KUKA KRL program: ps_604res_c1_orig.src, ps_604res_c1_orig.dat

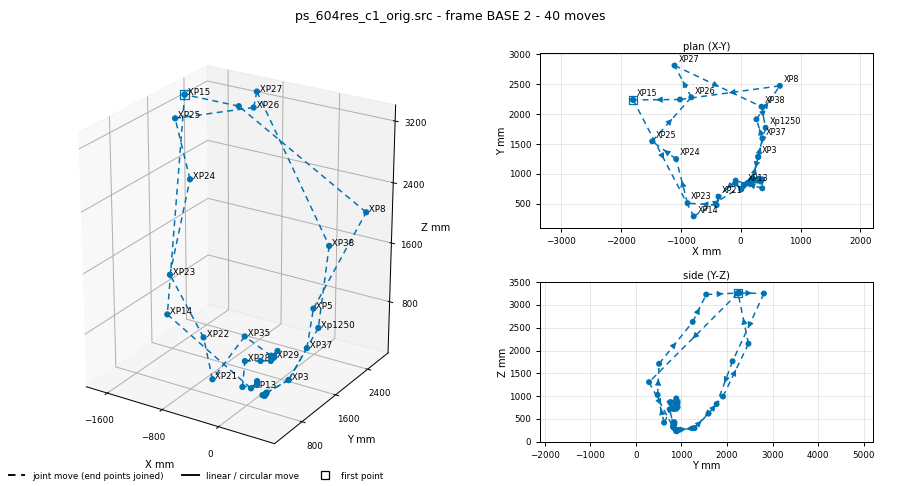
[picture p0: tool path of ps_604res_c1_orig.src in frame BASE 2, 40 of 40 moves have a stored position in this frame; points joined in program order, loops and branches not executed]
--- ps_604res_c1_orig.src ---
&ACCESS RVO
&COMMENT Solda Respot Accelo
DEF ps_604res_c1_orig( )
EXT e_Fraes1 ( )
EXT f_Fraes1 ( )
  ;FOLD INI;%{PE}%V2.2.2,%MKUKATPBASIS,%CINIT,%VCOMMON,%P
  ;FOLD BAS INI;%{PE}%V2.2.2,%MKUKATPBASIS,%CINIT,%VINIT,%P
  INTERRUPT DECL 3 WHEN $STOPMESS==TRUE DO IR_STOPM ( )
  INTERRUPT ON 3
  BAS (#INITMOV,0 )
  ;ENDFOLD
  ;FOLD A20 INI;%{E}%V2.2.2,%MKUKATPA20,%CINIT,%VINIT,%P
  IF ARC20==TRUE THEN
    A20 (ARC_INI)
    INTERRUPT DECL 6 WHEN $CYCFLAG[3]==FALSE DO A20(TECH_STOP2)
  ENDIF
  ;ENDFOLD
  ;FOLD A10 INI;%{E}%V2.2.2,%MKUKATPARC,%CINIT,%VINIT,%P
  IF A10_OPTION==#ACTIVE THEN
    INTERRUPT DECL 4 WHEN $CYCFLAG[2]==FALSE DO A10 (#APPL_ERROR)
    INTERRUPT DECL 7 WHEN A_ARC_SWI==#ACTIVE DO A10 (#ARC_SEAM)
    INTERRUPT DECL 5 WHEN A_FLY_ARC==TRUE DO A10 (#HPU_ARC)
    INTERRUPT  ON 5
    A10_INI ( )
  ENDIF
  ;ENDFOLD
  ;FOLD GRIPPER INI;%{E}%V2.2.2,%MKUKATPGRIPPER,%CINIT,%VINIT,%P
  USER_GRP(0,DUMMY,DUMMY,GDEFAULT)
  ;ENDFOLD
  ;FOLD SPOT INI;%{E}%V.2.2,%MKUKATPSPOT,%CINIT,%VINIT,%P
  USERSPOT(#INIT)
  ;ENDFOLD
  ;FOLD TOUCHSENSE INI;%{E}%V2.2.2,%MKUKATPTS,%CINIT,%VINIT,%P
  IF H70_OPTION THEN
    INTERRUPT DECL 15 WHEN $MEAS_PULSE[TOUCH_I[TOUCH_ACTIVE].IN_NR] DO H70 (6,CD0 )
    INTERRUPT DECL 16 WHEN $ZERO_MOVE DO H70 (7,CD0 )
    INTERRUPT DECL 17 WHEN $TECHPAR_C[FG_TOUCH,8]>0.5 DO H70 (8,CD0)
    H70 (1,CD0 )
  ENDIF
  ;ENDFOLD
  ;FOLD USER INI;%{P}%V2.2.2,%MKUKATPUSER,%CINIT,%VINIT,%P
  ;Make your modifications here
  ;ENDFOLD
  ;ENDFOLD

; Caracterização dos meios de produção: P13.060-R4
; Versão atual: 20/07/2013 12:00  Nome: Solda Respot Accelo
; Change: C1

chk_w1_wechs_ok ( )     ; VERIFICAÇÃO DE FERRAMENTA: C1

;FOLD Kollision.Ueberwachung_2_Ein ;%{PE}%MKUKATPUSER
COLLSTOP( 2, 1 ) ;INTERRUPTUEBERWACHT
;ENDFOLD

;FOLD PTP P15 CONT Vel= 80 % PDAT15 Tool[1]:GUN C1 Base[2]:Accelo;%{PE}%R 4.1.16,%MKUKATPBASIS,%CMOVE,%VPTP,%P 1:PTP, 2:P15, 3:C_PTP, 5:80, 7:PDAT15
$BWDSTART = FALSE
PDAT_ACT=PPDAT15
BAS(#PTP_DAT)
FDAT_ACT=FP15
BAS(#FRAMES)
BAS(#VEL_PTP,80)
PTP XP15 C_PTP
;ENDFOLD

;FOLD OUT 838 'Solic. Lib. Soldar Respot Geo1'  State= TRUE ;%{PE}%R 4.1.16,%MKUKATPBASIS,%COUT,%VOUTX,%P 2:838, 3:'Solic. Lib. Soldar Respot Geo1', 5:TRUE, 6:
$OUT[838]=TRUE
;ENDFOLD
;FOLD WAIT FOR IN 846 'R4 Aguarda Lib soldar RES geo 11'  State= TRUE ;%{PE}%R 4.1.16,%MKUKATPBASIS,%CWAIT_FOR,%VWAIT_FOR,%P 1:0, 2:846, 3:'R4 Aguarda Lib soldar RES geo 11', 5:TRUE, 6:
WAIT FOR $IN[846]==TRUE
;ENDFOLD
;FOLD OUT 838 'Solic. Lib. Soldar Respot Geo1'  State= FALSE ;%{PE}%R 4.1.16,%MKUKATPBASIS,%COUT,%VOUTX,%P 2:838, 3:'Solic. Lib. Soldar Respot Geo1', 5:FALSE, 6:
$OUT[838]=FALSE
;ENDFOLD


;FOLD OUT 851 'Libera AGV'  State= FALSE ;%{PE}%R 4.1.16,%MKUKATPBASIS,%COUT,%VOUTX,%P 2:851, 3:'Libera AGV', 5:FALSE, 6:
$OUT[851]=FALSE
;ENDFOLD


;FOLD PTP P14 CONT Vel= 80 % PDAT14 Tool[1]:GUN C1 Base[2]:Accelo;%{PE}%R 4.1.16,%MKUKATPBASIS,%CMOVE,%VPTP,%P 1:PTP, 2:P14, 3:C_PTP, 5:80, 7:PDAT14
$BWDSTART = FALSE
PDAT_ACT=PPDAT14
BAS(#PTP_DAT)
FDAT_ACT=FP14
BAS(#FRAMES)
BAS(#VEL_PTP,80)
PTP XP14 C_PTP
;ENDFOLD
;FOLD PTP P13 CONT Vel= 80 % PDAT13 Tool[1]:GUN C1 Base[2]:Accelo;%{PE}%R 4.1.16,%MKUKATPBASIS,%CMOVE,%VPTP,%P 1:PTP, 2:P13, 3:C_PTP, 5:80, 7:PDAT13
$BWDSTART = FALSE
PDAT_ACT=PPDAT13
BAS(#PTP_DAT)
FDAT_ACT=FP13
BAS(#FRAMES)
BAS(#VEL_PTP,80)
PTP XP13 C_PTP
;ENDFOLD
;FOLD PTP P17 CONT Vel= 80 % PDAT17 Tool[1]:GUN C1 Base[2]:Accelo;%{PE}%R 4.1.16,%MKUKATPBASIS,%CMOVE,%VPTP,%P 1:PTP, 2:P17, 3:C_PTP, 5:80, 7:PDAT17
$BWDSTART = FALSE
PDAT_ACT=PPDAT17
BAS(#PTP_DAT)
FDAT_ACT=FP17
BAS(#FRAMES)
BAS(#VEL_PTP,80)
PTP XP17 C_PTP
;ENDFOLD

;FOLD PTP SWP_62_0006 PDAT19 SPOT Gun= 1 RETR OPN PgNo1= 36 ACTIVE= 1 Tool[1]:GUN C1 Base[2]:Accelo;%{PE}%R 4.1.12,%MKUKATPSPOT,%CSPOT,%VPTP,%P 1:PTP, 2:SWP_62_0006, 3:, 5:80, 7:PDAT19, 10:1, 12:#FIRST, 14:#OPN, 16:36, 18:1, 20:0, 22:0, 24:1, 25:NORMAL
$BWDSTART = FALSE
PDAT_ACT=PPDAT19
BAS(#PTP_DAT)
FDAT_ACT=FSWP_62_0006
BAS(#FRAMES)
BAS(#VEL_PTP,PPDAT19.VEL)
S_ACT.GUN=1
S_ACT.PAIR=SDEFAULT.PAIR
S_ACT.RETR=#OPN
S_ACT.CLO_TM=1
S_ACT.PGNO1=36
S_ACT.PGNO2=SDEFAULT.PGNO2
S_ACT.PRESS1=SDEFAULT.PRESS1
S_ACT.PRESS2=SDEFAULT.PRESS2
S_READY=FALSE
PTP XSWP_62_0006
USERSPOT(#SPOT, S_ACT)
WAIT FOR S_READY
;ENDFOLD

;FOLD PTP P19 CONT Vel= 80 % PDAT20 Tool[1]:GUN C1 Base[2]:Accelo;%{PE}%R 4.1.16,%MKUKATPBASIS,%CMOVE,%VPTP,%P 1:PTP, 2:P19, 3:C_PTP, 5:80, 7:PDAT20
$BWDSTART = FALSE
PDAT_ACT=PPDAT20
BAS(#PTP_DAT)
FDAT_ACT=FP19
BAS(#FRAMES)
BAS(#VEL_PTP,80)
PTP XP19 C_PTP
;ENDFOLD
;FOLD PTP P20 CONT Vel= 80 % PDAT21 Tool[1]:GUN C1 Base[2]:Accelo;%{PE}%R 4.1.16,%MKUKATPBASIS,%CMOVE,%VPTP,%P 1:PTP, 2:P20, 3:C_PTP, 5:80, 7:PDAT21
$BWDSTART = FALSE
PDAT_ACT=PPDAT21
BAS(#PTP_DAT)
FDAT_ACT=FP20
BAS(#FRAMES)
BAS(#VEL_PTP,80)
PTP XP20 C_PTP
;ENDFOLD
;FOLD PTP P28  Vel= 80 % PDAT29 Tool[1]:GUN C1 Base[2]:Accelo;%{PE}%R 4.1.16,%MKUKATPBASIS,%CMOVE,%VPTP,%P 1:PTP, 2:P28, 3:, 5:80, 7:PDAT29
$BWDSTART = FALSE
PDAT_ACT=PPDAT29
BAS(#PTP_DAT)
FDAT_ACT=FP28
BAS(#FRAMES)
BAS(#VEL_PTP,80)
PTP XP28
;ENDFOLD
;FOLD PTP P30  Vel= 80 % PDAT31 Tool[1]:GUN C1 Base[2]:Accelo;%{PE}%R 4.1.16,%MKUKATPBASIS,%CMOVE,%VPTP,%P 1:PTP, 2:P30, 3:, 5:80, 7:PDAT31
$BWDSTART = FALSE
PDAT_ACT=PPDAT31
BAS(#PTP_DAT)
FDAT_ACT=FP30
BAS(#FRAMES)
BAS(#VEL_PTP,80)
PTP XP30
;ENDFOLD
;FOLD PTP P31  Vel= 80 % PDAT32 Tool[1]:GUN C1 Base[2]:Accelo;%{PE}%R 4.1.16,%MKUKATPBASIS,%CMOVE,%VPTP,%P 1:PTP, 2:P31, 3:, 5:80, 7:PDAT32
$BWDSTART = FALSE
PDAT_ACT=PPDAT32
BAS(#PTP_DAT)
FDAT_ACT=FP31
BAS(#FRAMES)
BAS(#VEL_PTP,80)
PTP XP31
;ENDFOLD
;FOLD PTP P29 PDAT30 SPOT Gun= 1 RETR OPN PgNo1= 1 ACTIVE= 1 Tool[1]:GUN C1 Base[2]:Accelo;%{PE}%R 4.1.12,%MKUKATPSPOT,%CSPOT,%VPTP,%P 1:PTP, 2:P29, 3:, 5:80, 7:PDAT30, 10:1, 12:#FIRST, 14:#OPN, 16:1, 18:1, 20:0, 22:0, 24:1, 25:NORMAL
$BWDSTART = FALSE
PDAT_ACT=PPDAT30
BAS(#PTP_DAT)
FDAT_ACT=FP29
BAS(#FRAMES)
BAS(#VEL_PTP,PPDAT30.VEL)
S_ACT.GUN=1
S_ACT.PAIR=SDEFAULT.PAIR
S_ACT.RETR=#OPN
S_ACT.CLO_TM=1
S_ACT.PGNO1=1
S_ACT.PGNO2=SDEFAULT.PGNO2
S_ACT.PRESS1=SDEFAULT.PRESS1
S_ACT.PRESS2=SDEFAULT.PRESS2
S_READY=FALSE
PTP XP29
USERSPOT(#SPOT, S_ACT)
WAIT FOR S_READY
;ENDFOLD
;FOLD PTP P36  Vel= 80 % PDAT37 Tool[1]:GUN C1 Base[2]:Accelo;%{PE}%R 4.1.16,%MKUKATPBASIS,%CMOVE,%VPTP,%P 1:PTP, 2:P36, 3:, 5:80, 7:PDAT37
$BWDSTART = FALSE
PDAT_ACT=PPDAT37
BAS(#PTP_DAT)
FDAT_ACT=FP36
BAS(#FRAMES)
BAS(#VEL_PTP,80)
PTP XP36
;ENDFOLD
;FOLD PTP P33 PDAT34 SPOT Gun= 1 RETR OPN PgNo1= 1 ACTIVE= 1 Tool[1]:GUN C1 Base[2]:Accelo;%{PE}%R 4.1.12,%MKUKATPSPOT,%CSPOT,%VPTP,%P 1:PTP, 2:P33, 3:, 5:80, 7:PDAT34, 10:1, 12:#FIRST, 14:#OPN, 16:1, 18:1, 20:0, 22:0, 24:1, 25:NORMAL
$BWDSTART = FALSE
PDAT_ACT=PPDAT34
BAS(#PTP_DAT)
FDAT_ACT=FP33
BAS(#FRAMES)
BAS(#VEL_PTP,PPDAT34.VEL)
S_ACT.GUN=1
S_ACT.PAIR=SDEFAULT.PAIR
S_ACT.RETR=#OPN
S_ACT.CLO_TM=1
S_ACT.PGNO1=1
S_ACT.PGNO2=SDEFAULT.PGNO2
S_ACT.PRESS1=SDEFAULT.PRESS1
S_ACT.PRESS2=SDEFAULT.PRESS2
S_READY=FALSE
PTP XP33
USERSPOT(#SPOT, S_ACT)
WAIT FOR S_READY
;ENDFOLD
;FOLD PTP P34  Vel= 80 % PDAT35 Tool[1]:GUN C1 Base[2]:Accelo;%{PE}%R 4.1.16,%MKUKATPBASIS,%CMOVE,%VPTP,%P 1:PTP, 2:P34, 3:, 5:80, 7:PDAT35
$BWDSTART = FALSE
PDAT_ACT=PPDAT35
BAS(#PTP_DAT)
FDAT_ACT=FP34
BAS(#FRAMES)
BAS(#VEL_PTP,80)
PTP XP34
;ENDFOLD
;FOLD PTP P35  Vel= 80 % PDAT36 Tool[1]:GUN C1 Base[2]:Accelo;%{PE}%R 4.1.16,%MKUKATPBASIS,%CMOVE,%VPTP,%P 1:PTP, 2:P35, 3:, 5:80, 7:PDAT36
$BWDSTART = FALSE
PDAT_ACT=PPDAT36
BAS(#PTP_DAT)
FDAT_ACT=FP35
BAS(#FRAMES)
BAS(#VEL_PTP,80)
PTP XP35
;ENDFOLD
;FOLD PTP P21 CONT Vel= 80 % PDAT22 Tool[1]:GUN C1 Base[2]:Accelo;%{PE}%R 4.1.16,%MKUKATPBASIS,%CMOVE,%VPTP,%P 1:PTP, 2:P21, 3:C_PTP, 5:80, 7:PDAT22
$BWDSTART = FALSE
PDAT_ACT=PPDAT22
BAS(#PTP_DAT)
FDAT_ACT=FP21
BAS(#FRAMES)
BAS(#VEL_PTP,80)
PTP XP21 C_PTP
;ENDFOLD
;FOLD PTP P22 CONT Vel= 80 % PDAT23 Tool[1]:GUN C1 Base[2]:Accelo;%{PE}%R 4.1.16,%MKUKATPBASIS,%CMOVE,%VPTP,%P 1:PTP, 2:P22, 3:C_PTP, 5:80, 7:PDAT23
$BWDSTART = FALSE
PDAT_ACT=PPDAT23
BAS(#PTP_DAT)
FDAT_ACT=FP22
BAS(#FRAMES)
BAS(#VEL_PTP,80)
PTP XP22 C_PTP
;ENDFOLD
;FOLD PTP P23 CONT Vel= 80 % PDAT24 Tool[1]:GUN C1 Base[2]:Accelo;%{PE}%R 4.1.16,%MKUKATPBASIS,%CMOVE,%VPTP,%P 1:PTP, 2:P23, 3:C_PTP, 5:80, 7:PDAT24
$BWDSTART = FALSE
PDAT_ACT=PPDAT24
BAS(#PTP_DAT)
FDAT_ACT=FP23
BAS(#FRAMES)
BAS(#VEL_PTP,80)
PTP XP23 C_PTP
;ENDFOLD
;FOLD PTP P24 CONT Vel= 80 % PDAT25 Tool[1]:GUN C1 Base[2]:Accelo;%{PE}%R 4.1.16,%MKUKATPBASIS,%CMOVE,%VPTP,%P 1:PTP, 2:P24, 3:C_PTP, 5:80, 7:PDAT25
$BWDSTART = FALSE
PDAT_ACT=PPDAT25
BAS(#PTP_DAT)
FDAT_ACT=FP24
BAS(#FRAMES)
BAS(#VEL_PTP,80)
PTP XP24 C_PTP
;ENDFOLD
;FOLD PTP P25 CONT Vel= 80 % PDAT26 Tool[1]:GUN C1 Base[2]:Accelo;%{PE}%R 4.1.16,%MKUKATPBASIS,%CMOVE,%VPTP,%P 1:PTP, 2:P25, 3:C_PTP, 5:80, 7:PDAT26
$BWDSTART = FALSE
PDAT_ACT=PPDAT26
BAS(#PTP_DAT)
FDAT_ACT=FP25
BAS(#FRAMES)
BAS(#VEL_PTP,80)
PTP XP25 C_PTP
;ENDFOLD
;FOLD PTP P26 CONT Vel= 80 % PDAT27 Tool[1]:GUN C1 Base[2]:Accelo;%{PE}%R 4.1.16,%MKUKATPBASIS,%CMOVE,%VPTP,%P 1:PTP, 2:P26, 3:C_PTP, 5:80, 7:PDAT27
$BWDSTART = FALSE
PDAT_ACT=PPDAT27
BAS(#PTP_DAT)
FDAT_ACT=FP26
BAS(#FRAMES)
BAS(#VEL_PTP,80)
PTP XP26 C_PTP
;ENDFOLD
;FOLD PTP P27 CONT Vel= 80 % PDAT28 Tool[1]:GUN C1 Base[2]:Accelo;%{PE}%R 4.1.16,%MKUKATPBASIS,%CMOVE,%VPTP,%P 1:PTP, 2:P27, 3:C_PTP, 5:80, 7:PDAT28
$BWDSTART = FALSE
PDAT_ACT=PPDAT28
BAS(#PTP_DAT)
FDAT_ACT=FP27
BAS(#FRAMES)
BAS(#VEL_PTP,80)
PTP XP27 C_PTP
;ENDFOLD
;FOLD PTP P38 CONT Vel= 80 % PDAT39 Tool[1]:GUN C1 Base[2]:Accelo;%{PE}%R 4.1.16,%MKUKATPBASIS,%CMOVE,%VPTP,%P 1:PTP, 2:P38, 3:C_PTP, 5:80, 7:PDAT39
$BWDSTART = FALSE
PDAT_ACT=PPDAT39
BAS(#PTP_DAT)
FDAT_ACT=FP38
BAS(#FRAMES)
BAS(#VEL_PTP,80)
PTP XP38 C_PTP
;ENDFOLD
;FOLD PTP p1250 CONT Vel= 90 % P_OLP4 Tool[1]:GUN C1 Base[2]:Accelo;%{PE}%R 4.1.16,%MKUKATPBASIS,%CMOVE,%VPTP,%P 1:PTP, 2:p1250, 3:C_PTP, 5:90, 7:P_OLP4
$BWDSTART = FALSE
PDAT_ACT=PP_OLP4
BAS(#PTP_DAT)
FDAT_ACT=Fp1250
BAS(#FRAMES)
BAS(#VEL_PTP,90)
PTP Xp1250 C_PTP
;ENDFOLD
;FOLD PTP P3 CONT Vel= 90 % PDAT4 Tool[1]:GUN C1 Base[2]:Accelo;%{PE}%R 4.1.16,%MKUKATPBASIS,%CMOVE,%VPTP,%P 1:PTP, 2:P3, 3:C_PTP, 5:90, 7:PDAT4
$BWDSTART = FALSE
PDAT_ACT=PPDAT4
BAS(#PTP_DAT)
FDAT_ACT=FP3
BAS(#FRAMES)
BAS(#VEL_PTP,90)
PTP XP3 C_PTP
;ENDFOLD
;FOLD PTP p1255 CONT Vel= 80 % P_OLP9 Tool[1]:GUN C1 Base[2]:Accelo;%{PE}%R 4.1.16,%MKUKATPBASIS,%CMOVE,%VPTP,%P 1:PTP, 2:p1255, 3:C_PTP, 5:80, 7:P_OLP9
$BWDSTART = FALSE
PDAT_ACT=PP_OLP9
BAS(#PTP_DAT)
FDAT_ACT=Fp1255
BAS(#FRAMES)
BAS(#VEL_PTP,80)
PTP Xp1255 C_PTP
;ENDFOLD
;FOLD PTP p1256  Vel= 60 % P_OLP10 Tool[1]:GUN C1 Base[2]:Accelo;%{PE}%R 4.1.16,%MKUKATPBASIS,%CMOVE,%VPTP,%P 1:PTP, 2:p1256, 3:, 5:60, 7:P_OLP10
$BWDSTART = FALSE
PDAT_ACT=PP_OLP10
BAS(#PTP_DAT)
FDAT_ACT=Fp1256
BAS(#FRAMES)
BAS(#VEL_PTP,60)
PTP Xp1256
;ENDFOLD

;FOLD OUT 848 'Area de Solda'  State= FALSE ;%{PE}%R 4.1.16,%MKUKATPBASIS,%COUT,%VOUTX,%P 2:848, 3:'Area de Solda', 5:FALSE, 6:
$OUT[848]=FALSE
;ENDFOLD

;FOLD ; comeco solda;%{PE}%R 4.1.16,%MKUKATPBASIS,%CCOMMENT,%VNORMAL,%P 2:comeco solda
;ENDFOLD
;FOLD OUT 839 'R4 Soldando'  State= TRUE ;%{PE}%R 4.1.16,%MKUKATPBASIS,%COUT,%VOUTX,%P 2:839, 3:'R4 Soldando', 5:TRUE, 6:
$OUT[839]=TRUE
;ENDFOLD

;FOLD PTP p1257 CONT Vel= 60 % PDAT40 Tool[1]:GUN C1 Base[2]:Accelo;%{PE}%R 4.1.16,%MKUKATPBASIS,%CMOVE,%VPTP,%P 1:PTP, 2:p1257, 3:C_PTP, 5:60, 7:PDAT40
$BWDSTART = FALSE
PDAT_ACT=PPDAT40
BAS(#PTP_DAT)
FDAT_ACT=Fp1257
BAS(#FRAMES)
BAS(#VEL_PTP,60)
PTP Xp1257 C_PTP
;ENDFOLD

;FOLD ; SWP_60_0214;%{PE}%R2.2,%MKUKATPBASIS,%CCOMMENT,%VNORMAL,%P 2: SWP_60_0214
;ENDFOLD
;FOLD LIN P2 CPDAT1 SPOT Gun= 1 RETR OPN PgNo1= 14 ACTIVE= 1 Tool[1]:GUN C1 Base[2]:Accelo;%{PE}%R 4.1.12,%MKUKATPSPOT,%CSPOT,%VLIN,%P 1:LIN, 2:P2, 3:, 5:2, 7:CPDAT1, 10:1, 12:#FIRST, 14:#OPN, 16:14, 18:1, 20:0, 22:0, 24:1, 25:NORMAL
$BWDSTART = FALSE
LDAT_ACT=LCPDAT1
BAS(#CP_DAT)
FDAT_ACT=FP2
BAS(#FRAMES)
BAS(#VEL_CP,LCPDAT1.VEL)
S_ACT.GUN=1
S_ACT.PAIR=SDEFAULT.PAIR
S_ACT.RETR=#OPN
S_ACT.CLO_TM=1
S_ACT.PGNO1=14
S_ACT.PGNO2=SDEFAULT.PGNO2
S_ACT.PRESS1=SDEFAULT.PRESS1
S_ACT.PRESS2=SDEFAULT.PRESS2
S_READY=FALSE
LIN XP2
USERSPOT(#SPOT, S_ACT)
WAIT FOR S_READY
;ENDFOLD

;FOLD ; SWP_60_0216;%{PE}%R2.2,%MKUKATPBASIS,%CCOMMENT,%VNORMAL,%P 2: SWP_60_0216
;ENDFOLD
;FOLD LIN P4 CPDAT3 SPOT Gun= 1 RETR OPN PgNo1= 15 ACTIVE= 1 Tool[1]:GUN C1 Base[2]:Accelo;%{PE}%R 4.1.12,%MKUKATPSPOT,%CSPOT,%VLIN,%P 1:LIN, 2:P4, 3:, 5:2, 7:CPDAT3, 10:1, 12:#FIRST, 14:#OPN, 16:15, 18:1, 20:0, 22:0, 24:1, 25:NORMAL
$BWDSTART = FALSE
LDAT_ACT=LCPDAT3
BAS(#CP_DAT)
FDAT_ACT=FP4
BAS(#FRAMES)
BAS(#VEL_CP,LCPDAT3.VEL)
S_ACT.GUN=1
S_ACT.PAIR=SDEFAULT.PAIR
S_ACT.RETR=#OPN
S_ACT.CLO_TM=1
S_ACT.PGNO1=15
S_ACT.PGNO2=SDEFAULT.PGNO2
S_ACT.PRESS1=SDEFAULT.PRESS1
S_ACT.PRESS2=SDEFAULT.PRESS2
S_READY=FALSE
LIN XP4
USERSPOT(#SPOT, S_ACT)
WAIT FOR S_READY
;ENDFOLD

;FOLD LIN p2  Vel= 0.4 m/s CPDAT4 Tool[1]:GUN C1 Base[2]:Accelo;%{PE}%R 4.1.16,%MKUKATPBASIS,%CMOVE,%VLIN,%P 1:LIN, 2:p2, 3:, 5:0.4, 7:CPDAT4
$BWDSTART = FALSE
LDAT_ACT=LCPDAT4
BAS(#CP_DAT)
FDAT_ACT=Fp2
BAS(#FRAMES)
BAS(#VEL_CP,0.4)
LIN Xp2
;ENDFOLD

;FOLD OUT 839 'R4 Soldando'  State= FALSE ;%{PE}%R 4.1.16,%MKUKATPBASIS,%COUT,%VOUTX,%P 2:839, 3:'R4 Soldando', 5:FALSE, 6:
$OUT[839]=FALSE
;ENDFOLD
;FOLD OUT 848 'Area de Solda'  State= TRUE ;%{PE}%R 4.1.16,%MKUKATPBASIS,%COUT,%VOUTX,%P 2:848, 3:'Area de Solda', 5:TRUE, 6:
$OUT[848]=TRUE
;ENDFOLD

;FOLD LIN p1257 CONT Vel= 0.5 m/s CPDAT5 Tool[1]:GUN C1 Base[2]:Accelo;%{PE}%R 4.1.16,%MKUKATPBASIS,%CMOVE,%VLIN,%P 1:LIN, 2:p1257, 3:C_DIS, 5:0.5, 7:CPDAT5
$BWDSTART = FALSE
LDAT_ACT=LCPDAT5
BAS(#CP_DAT)
FDAT_ACT=Fp1257
BAS(#FRAMES)
BAS(#VEL_CP,0.5)
LIN Xp1257 C_DIS
;ENDFOLD

;FOLD PTP p1256 CONT Vel= 70 % P_OLP16 Tool[1]:GUN C1 Base[2]:Accelo;%{PE}%R 4.1.16,%MKUKATPBASIS,%CMOVE,%VPTP,%P 1:PTP, 2:p1256, 3:C_PTP, 5:70, 7:P_OLP16
$BWDSTART = FALSE
PDAT_ACT=PP_OLP16
BAS(#PTP_DAT)
FDAT_ACT=Fp1256
BAS(#FRAMES)
BAS(#VEL_PTP,70)
PTP Xp1256 C_PTP
;ENDFOLD
;FOLD PTP p1255 CONT Vel= 90 % P_OLP17 Tool[1]:GUN C1 Base[2]:Accelo;%{PE}%R 4.1.16,%MKUKATPBASIS,%CMOVE,%VPTP,%P 1:PTP, 2:p1255, 3:C_PTP, 5:90, 7:P_OLP17
$BWDSTART = FALSE
PDAT_ACT=PP_OLP17
BAS(#PTP_DAT)
FDAT_ACT=Fp1255
BAS(#FRAMES)
BAS(#VEL_PTP,90)
PTP Xp1255 C_PTP
;ENDFOLD
;FOLD PTP p3 CONT Vel= 90 % P_OLP18 Tool[1]:GUN C1 Base[2]:Accelo;%{PE}%R 4.1.16,%MKUKATPBASIS,%CMOVE,%VPTP,%P 1:PTP, 2:p3, 3:C_PTP, 5:90, 7:P_OLP18
$BWDSTART = FALSE
PDAT_ACT=PP_OLP18
BAS(#PTP_DAT)
FDAT_ACT=Fp3
BAS(#FRAMES)
BAS(#VEL_PTP,90)
PTP Xp3 C_PTP
;ENDFOLD
;FOLD PTP P37 CONT Vel= 90 % PDAT38 Tool[1]:GUN C1 Base[2]:Accelo;%{PE}%R 4.1.16,%MKUKATPBASIS,%CMOVE,%VPTP,%P 1:PTP, 2:P37, 3:C_PTP, 5:90, 7:PDAT38
$BWDSTART = FALSE
PDAT_ACT=PPDAT38
BAS(#PTP_DAT)
FDAT_ACT=FP37
BAS(#FRAMES)
BAS(#VEL_PTP,90)
PTP XP37 C_PTP
;ENDFOLD
;FOLD PTP P5 CONT Vel= 90 % PDAT5 Tool[1]:GUN C1 Base[2]:Accelo;%{PE}%R 4.1.16,%MKUKATPBASIS,%CMOVE,%VPTP,%P 1:PTP, 2:P5, 3:C_PTP, 5:90, 7:PDAT5
$BWDSTART = FALSE
PDAT_ACT=PPDAT5
BAS(#PTP_DAT)
FDAT_ACT=FP5
BAS(#FRAMES)
BAS(#VEL_PTP,90)
PTP XP5 C_PTP
;ENDFOLD
;FOLD PTP P8 CONT Vel= 90 % PDAT8 Tool[1]:GUN C1 Base[2]:Accelo;%{PE}%R 4.1.16,%MKUKATPBASIS,%CMOVE,%VPTP,%P 1:PTP, 2:P8, 3:C_PTP, 5:90, 7:PDAT8
$BWDSTART = FALSE
PDAT_ACT=PPDAT8
BAS(#PTP_DAT)
FDAT_ACT=FP8
BAS(#FRAMES)
BAS(#VEL_PTP,90)
PTP XP8 C_PTP
;ENDFOLD
;FOLD PTP P16  Vel= 80 % PDAT16 Tool[1]:GUN C1 Base[2]:Accelo;%{PE}%R 4.1.16,%MKUKATPBASIS,%CMOVE,%VPTP,%P 1:PTP, 2:P16, 3:, 5:80, 7:PDAT16
$BWDSTART = FALSE
PDAT_ACT=PPDAT16
BAS(#PTP_DAT)
FDAT_ACT=FP16
BAS(#FRAMES)
BAS(#VEL_PTP,80)
PTP XP16
;ENDFOLD

;FOLD PULSE 846 'R4 solda RES geo1 concluida'  State= TRUE CONT  Time= 3 sec;%{PE}%R 4.1.16,%MKUKATPBASIS,%COUT,%VPULSE,%P 2:846, 3:'R4 solda RES geo1 concluida', 5:TRUE, 6:CONTINUE, 8:3
CONTINUE
PULSE($OUT[846], TRUE,3)
;ENDFOLD

;FOLD ; END INTERLOCK COM R2;%{PE}%R 4.1.16,%MKUKATPBASIS,%CCOMMENT,%VNORMAL,%P 2:END INTERLOCK COM R2
;ENDFOLD
;FOLD Kollision.Ueberwachung_2_Aus ;%{PE}%MKUKATPUSER
COLLSTOP( 2, 2 )
;ENDFOLD

;FOLD ; START INTERLOCK R3;%{PE}%R 4.1.16,%MKUKATPBASIS,%CCOMMENT,%VNORMAL,%P 2:START INTERLOCK R3
;ENDFOLD
;FOLD Kollision.Ueberwachung_3_Aus ;%{PE}%MKUKATPUSER
COLLSTOP( 3, 2 )
;ENDFOLD

;FOLD PTP p1271 CONT Vel= 90 % P_OLP25 Tool[1]:GUN C1 Base[2]:Accelo;%{PE}%R 4.1.16,%MKUKATPBASIS,%CMOVE,%VPTP,%P 1:PTP, 2:p1271, 3:C_PTP, 5:90, 7:P_OLP25
$BWDSTART = FALSE
PDAT_ACT=PP_OLP25
BAS(#PTP_DAT)
FDAT_ACT=Fp1271
BAS(#FRAMES)
BAS(#VEL_PTP,90)
PTP Xp1271 C_PTP
;ENDFOLD

END

--- ps_604res_c1_orig.dat ---
&ACCESS RVO
&COMMENT Solda Respot Accelo
DEFDAT ps_604res_c1_orig
;FOLD EXTERNAL DECLARATIONS;%{PE}%V2.2.2,%MKUKATPBASIS,%CEXT,%VCOMMON,%P
;FOLD BAS EXT;%{PE}%V2.2.2,%MKUKATPBASIS,%CEXT,%VEXT,%P
EXT  BAS (BAS_COMMAND  :IN,REAL  :IN )
DECL INT SUCCESS
;ENDFOLD
;FOLD A10 EXT;%{E}%V2.2.2,%MKUKATPARC,%CEXT,%VEXT,%P
EXT  A10 (A_CMD_T  :IN,A_STRT_T  :IN,A_WELD_T  :IN,A_END_T  :IN,INT  :IN )
;ENDFOLD
;FOLD A20 EXT;%{E}%V2.2.2,%MKUKATPA20,%CEXT,%VEXT,%P
EXT  A20 (INT  :IN,WELD_ST  :IN,WELD_FI  :IN,INT  :IN )
;ENDFOLD
;FOLD GRIPPER EXT;%{E}%V2.2.2,%MKUKATPGRIPPER,%CEXT,%VEXT,%P
EXT  H50 (INT  :IN,INT  :IN,INT  :IN,GRP_TYP  :IN )
;ENDFOLD
;FOLD SPOT EXT;%{E}%V2.2.2,%MKUKATPSPOT,%CEXT,%VEXT,%P
EXT  USERSPOT (S_COMMAND  :IN,SPOT_TYPE  :IN )
;ENDFOLD
;FOLD TOUCHSENSE EXT;%{E}%V2.2.2,%MKUKATPTS,%CEXT,%VEXT,%P
EXT  H70 (INT  :IN,SRCH_TYP_2  :OUT,E6POS  :IN,SRCH_TYP_3  :IN,SRCH_TYP_2  :IN,SRCH_TYP_2  :IN,SRCH_TYP_2  :IN,SRCH_TYP_2  :IN,SRCH_TYP_2  :IN,INT  :IN )
;ENDFOLD
;FOLD USER EXT;%{}%V2.2.2,%MKUKATPUSER,%CEXT,%VEXT,%P
;Make here your modifications
;ENDFOLD
;ENDFOLD

;# ============ START PATH : swp_p13060r4_ltc_resp1_c1 =============
DECL FDAT Fp1250={TOOL_NO 1,BASE_NO 2,IPO_FRAME #BASE}
DECL PDAT PP_OLP4={VEL 100.0,ACC 100.0,APO_DIST 10.0}
DECL E6POS Xp1250={x 416.153503,y 1772.771,z 826.273682,a 22.6149693,b 41.6934814,c -97.8162537,s 6,t 59,e1 0.0,e2 0.0,e3 0.0,e4 0.0,e5 0.0,e6 0.0}
DECL FDAT Fp1255={TOOL_NO 1,BASE_NO 2,IPO_FRAME #BASE}
DECL PDAT PP_OLP9={VEL 100.0,ACC 100.0,APO_DIST 10.0}
DECL E6POS Xp1255={x 201.438705,y 923.264893,z 259.861908,a -0.494082987,b 36.3943787,c -77.2345734,s 6,t 59,e1 0.0,e2 0.0,e3 0.0,e4 0.0,e5 0.0,e6 0.0}
DECL FDAT Fp1256={TOOL_NO 1,BASE_NO 2,IPO_FRAME #BASE}
DECL PDAT PP_OLP10={VEL 100.0,ACC 100.0,APO_DIST 100.0}
DECL E6POS Xp1256={x 199.555206,y 905.03717,z 250.693405,a -2.2262361,b 39.3286095,c -77.6910934,s 6,t 59,e1 0.0,e2 0.0,e3 0.0,e4 0.0,e5 0.0,e6 0.0}
DECL FDAT Fp1257={TOOL_NO 1,BASE_NO 2,IPO_FRAME #BASE}
DECL E6POS Xp1257={x 201.019608,y 901.876587,z 248.831894,a -3.6396811,b 37.6043892,c -79.63694,s 6,t 59,e1 0.0,e2 0.0,e3 0.0,e4 0.0,e5 0.0,e6 0.0}
DECL PDAT PP_OLP16={VEL 100.0,ACC 100.0,APO_DIST 100.0}
DECL PDAT PP_OLP17={VEL 100.0,ACC 100.0,APO_DIST 100.0}
DECL PDAT PP_OLP18={VEL 100.0,ACC 100.0,APO_DIST 100.0}
DECL FDAT Fp1271={TOOL_NO 1,BASE_NO 2,IPO_FRAME #BASE}
DECL PDAT PP_OLP25={VEL 100.0,ACC 100.0,APO_DIST 100.0}
DECL E6POS Xp1271={x -1796.38599,y 2237.50098,z 3255.19995,a 90.0,b 0.0,c -170.0,s 6,t 18}
DECL BASIS_SUGG_T LAST_BASIS={POINT1[] "P38                     ",POINT2[] "P38                     ",CP_PARAMS[] "CPDAT3                  ",PTP_PARAMS[] "PDAT39                  ",CONT[] "C_PTP                   ",CP_VEL[] "2                       ",PTP_VEL[] "80                      "}
DECL E6POS XP2={x 192.499405,y 894.710571,z 231.026505,a -2.51362205,b 57.5632896,c -90.971283,s 6,t 59,e1 0.0,e2 0.0,e3 0.0,e4 0.0,e5 0.0,e6 0.0}
DECL FDAT FP2={TOOL_NO 1,BASE_NO 2,IPO_FRAME #BASE}
DECL LDAT LCPDAT1={VEL 0.400000006,ACC 100.0,APO_DIST 100.0,APO_FAC 50.0}
DECL E6POS XP3={x 293.535309,y 1285.255,z 298.4841,a 19.5087795,b 37.8742714,c -66.1795578,s 6,t 59,e1 0.0,e2 0.0,e3 0.0,e4 0.0,e5 0.0,e6 0.0}
DECL FDAT FP3={TOOL_NO 1,BASE_NO 2,IPO_FRAME #BASE}
DECL PDAT PPDAT4={VEL 100.0,ACC 100.0,APO_DIST 100.0}
DECL E6POS XP4={x 164.863205,y 892.523071,z 233.009293,a -179.284607,b 77.8195572,c 92.4647827,s 6,t 59,e1 0.0,e2 0.0,e3 0.0,e4 0.0,e5 0.0,e6 0.0}
DECL FDAT FP4={TOOL_NO 1,BASE_NO 2,IPO_FRAME #BASE}
DECL LDAT LCPDAT3={VEL 0.400000006,ACC 100.0,APO_DIST 100.0,APO_FAC 50.0}
DECL LDAT LCPDAT4={VEL 2.0,ACC 100.0,APO_DIST 100.0,APO_FAC 50.0}
DECL LDAT LCPDAT5={VEL 2.0,ACC 100.0,APO_DIST 0.0,APO_FAC 50.0}
DECL E6POS XP5={x 263.258087,y 1912.71802,z 991.068176,a 29.9836006,b 37.9695091,c -91.8605194,s 6,t 59,e1 0.0,e2 0.0,e3 0.0,e4 0.0,e5 0.0,e6 0.0}
DECL FDAT FP5={TOOL_NO 1,BASE_NO 2,IPO_FRAME #BASE}
DECL PDAT PPDAT5={VEL 100.0,ACC 100.0,APO_DIST 100.0}
DECL E6POS XP8={x 654.817688,y 2472.11597,z 2149.81592,a -6.18557692,b 40.8391304,c -163.516998,s 6,t 59,e1 0.0,e2 0.0,e3 0.0,e4 0.0,e5 0.0,e6 0.0}
DECL FDAT FP8={TOOL_NO 1,BASE_NO 2,IPO_FRAME #BASE}
DECL PDAT PPDAT8={VEL 100.0,ACC 100.0,APO_DIST 100.0}
DECL E6POS XP13={x 50.1561012,y 814.575012,z 327.331787,a -23.4693108,b -63.3067894,c 9.10689068,s 6,t 19,e1 0.0,e2 0.0,e3 0.0,e4 0.0,e5 0.0,e6 0.0}
DECL FDAT FP13={TOOL_NO 1,BASE_NO 2,IPO_FRAME #BASE}
DECL PDAT PPDAT13={VEL 100.0,ACC 80.0,APO_DIST 100.0}
DECL E6POS XP14={x -784.374512,y 291.430389,z 1307.67896,a -157.717606,b -64.2434464,c 123.140198,s 6,t 18,e1 0.0,e2 0.0,e3 0.0,e4 0.0,e5 0.0,e6 0.0}
DECL FDAT FP14={TOOL_NO 1,BASE_NO 2,IPO_FRAME #BASE}
DECL PDAT PPDAT14={VEL 100.0,ACC 80.0,APO_DIST 100.0}
DECL E6POS XP15={x -1796.38403,y 2237.50293,z 3255.19995,a 89.9999695,b 2.24131709E-05,c -170.0,s 6,t 18,e1 0.0,e2 0.0,e3 0.0,e4 0.0,e5 0.0,e6 0.0}
DECL FDAT FP15={TOOL_NO 1,BASE_NO 2,IPO_FRAME #BASE}
DECL PDAT PPDAT15={VEL 100.0,ACC 80.0,APO_DIST 100.0}
DECL E6POS XP16={x -1013.565,y 2243.53003,z 3255.20093,a -69.9993134,b 8.53213442E-06,c -170.0,s 6,t 27,e1 0.0,e2 0.0,e3 0.0,e4 0.0,e5 0.0,e6 0.0}
DECL FDAT FP16={TOOL_NO 1,BASE_NO 2,IPO_FRAME #BASE}
DECL PDAT PPDAT16={VEL 100.0,ACC 80.0,APO_DIST 100.0}
DECL E6POS XP17={x 117.853996,y 845.772278,z 407.121887,a -27.4254494,b -71.2756577,c 21.1497192,s 6,t 19,e1 0.0,e2 0.0,e3 0.0,e4 0.0,e5 0.0,e6 0.0}
DECL FDAT FP17={TOOL_NO 1,BASE_NO 2,IPO_FRAME #BASE}
DECL PDAT PPDAT17={VEL 100.0,ACC 80.0,APO_DIST 100.0}
DECL PDAT PPDAT19={VEL 60.0,ACC 100.0,APO_DIST 100.0}
DECL E6POS XP19={x 117.692101,y 844.877991,z 377.491089,a -23.7453804,b -65.4931717,c 14.1894503,s 6,t 19,e1 0.0,e2 0.0,e3 0.0,e4 0.0,e5 0.0,e6 0.0}
DECL FDAT FP19={TOOL_NO 1,BASE_NO 2,IPO_FRAME #BASE}
DECL PDAT PPDAT20={VEL 100.0,ACC 80.0,APO_DIST 100.0}
DECL E6POS XP20={x -85.7270126,y 841.264709,z 296.153412,a -23.7463799,b -65.4932327,c 14.19063,s 6,t 19,e1 0.0,e2 0.0,e3 0.0,e4 0.0,e5 0.0,e6 0.0}
DECL FDAT FP20={TOOL_NO 1,BASE_NO 2,IPO_FRAME #BASE}
DECL PDAT PPDAT21={VEL 100.0,ACC 80.0,APO_DIST 100.0}
DECL E6POS XP21={x -370.383789,y 620.823975,z 418.002502,a -35.7969093,b -70.3211136,c 12.5743704,s 6,t 18,e1 0.0,e2 0.0,e3 0.0,e4 0.0,e5 0.0,e6 0.0}
DECL FDAT FP21={TOOL_NO 1,BASE_NO 2,IPO_FRAME #BASE}
DECL PDAT PPDAT22={VEL 100.0,ACC 80.0,APO_DIST 100.0}
DECL E6POS XP22={x -400.706787,y 479.283295,z 1027.30505,a -143.368393,b -83.5602112,c 113.175903,s 6,t 18,e1 0.0,e2 0.0,e3 0.0,e4 0.0,e5 0.0,e6 0.0}
DECL FDAT FP22={TOOL_NO 1,BASE_NO 2,IPO_FRAME #BASE}
DECL PDAT PPDAT23={VEL 100.0,ACC 80.0,APO_DIST 100.0}
DECL E6POS XP23={x -888.394287,y 511.849213,z 1710.35706,a 150.920593,b -61.3315392,c 169.039703,s 6,t 18,e1 0.0,e2 0.0,e3 0.0,e4 0.0,e5 0.0,e6 0.0}
DECL FDAT FP23={TOOL_NO 1,BASE_NO 2,IPO_FRAME #BASE}
DECL PDAT PPDAT24={VEL 100.0,ACC 80.0,APO_DIST 100.0}
DECL E6POS XP24={x -1077.47095,y 1248.70398,z 2628.5249,a 158.721298,b -22.2133102,c -174.973297,s 6,t 18,e1 0.0,e2 0.0,e3 0.0,e4 0.0,e5 0.0,e6 0.0}
DECL FDAT FP24={TOOL_NO 1,BASE_NO 2,IPO_FRAME #BASE}
DECL PDAT PPDAT25={VEL 100.0,ACC 80.0,APO_DIST 100.0}
DECL E6POS XP25={x -1478.28003,y 1545.23706,z 3228.60693,a 176.167297,b -0.158624604,c -177.060303,s 6,t 19,e1 0.0,e2 0.0,e3 0.0,e4 0.0,e5 0.0,e6 0.0}
DECL FDAT FP25={TOOL_NO 1,BASE_NO 2,IPO_FRAME #BASE}
DECL PDAT PPDAT26={VEL 100.0,ACC 80.0,APO_DIST 100.0}
DECL E6POS XP26={x -824.532227,y 2279.98901,z 3263.74707,a -148.510101,b -15.7248497,c -172.654694,s 6,t 19,e1 0.0,e2 0.0,e3 0.0,e4 0.0,e5 0.0,e6 0.0}
DECL FDAT FP26={TOOL_NO 1,BASE_NO 2,IPO_FRAME #BASE}
DECL PDAT PPDAT27={VEL 100.0,ACC 80.0,APO_DIST 100.0}
DECL E6POS XP27={x -1105.05396,y 2811.37988,z 3251.24512,a -99.2128296,b -16.5289497,c -173.276001,s 6,t 19,e1 0.0,e2 0.0,e3 0.0,e4 0.0,e5 0.0,e6 0.0}
DECL FDAT FP27={TOOL_NO 1,BASE_NO 2,IPO_FRAME #BASE}
DECL PDAT PPDAT28={VEL 100.0,ACC 80.0,APO_DIST 100.0}
DECL E6POS XSWP_62_0006={x 117.328201,y 845.899292,z 429.122314,a -23.7451897,b -65.4931412,c 14.1892204,s 6,t 19,e1 0.0,e2 0.0,e3 0.0,e4 0.0,e5 0.0,e6 0.0}
DECL FDAT FSWP_62_0006={TOOL_NO 1,BASE_NO 2,IPO_FRAME #BASE}
DECL E6POS XP28={x 9.95831108,y 743.330322,z 711.825684,a 35.4068489,b -57.6428719,c -39.2142601,s 6,t 19,e1 0.0,e2 0.0,e3 0.0,e4 0.0,e5 0.0,e6 0.0}
DECL FDAT FP28={TOOL_NO 1,BASE_NO 2,IPO_FRAME #BASE}
DECL PDAT PPDAT29={VEL 100.0,ACC 100.0,APO_DIST 100.0}
DECL E6POS XP29={x 303.400696,y 919.1203,z 759.304016,a 61.3300209,b -15.7221203,c -62.2064285,s 6,t 19,e1 0.0,e2 0.0,e3 0.0,e4 0.0,e5 0.0,e6 0.0}
DECL FDAT FP29={TOOL_NO 1,BASE_NO 2,IPO_FRAME #BASE}
DECL PDAT PPDAT30={VEL 60.0,ACC 100.0,APO_DIST 100.0}
DECL E6POS XP30={x 168.876007,y 837.242188,z 716.171326,a 51.3181686,b -36.4406509,c -52.901989,s 6,t 19,e1 0.0,e2 0.0,e3 0.0,e4 0.0,e5 0.0,e6 0.0}
DECL FDAT FP30={TOOL_NO 1,BASE_NO 2,IPO_FRAME #BASE}
DECL PDAT PPDAT31={VEL 100.0,ACC 100.0,APO_DIST 100.0}
DECL E6POS XP31={x 279.768585,y 889.198975,z 723.528625,a 57.8372498,b -23.8768005,c -58.8607216,s 6,t 19,e1 0.0,e2 0.0,e3 0.0,e4 0.0,e5 0.0,e6 0.0}
DECL FDAT FP31={TOOL_NO 1,BASE_NO 2,IPO_FRAME #BASE}
DECL PDAT PPDAT32={VEL 100.0,ACC 100.0,APO_DIST 100.0}
DECL E6POS XP33={x 359.795288,y 910.380127,z 867.386902,a 57.8205719,b -24.4404907,c -59.7361984,s 6,t 19,e1 0.0,e2 0.0,e3 0.0,e4 0.0,e5 0.0,e6 0.0}
DECL FDAT FP33={TOOL_NO 1,BASE_NO 2,IPO_FRAME #BASE}
DECL PDAT PPDAT34={VEL 60.0,ACC 100.0,APO_DIST 100.0}
DECL E6POS XP34={x 361.277802,y 759.951477,z 870.37738,a 57.8207092,b -24.4404297,c -59.7361908,s 6,t 19,e1 0.0,e2 0.0,e3 0.0,e4 0.0,e5 0.0,e6 0.0}
DECL FDAT FP34={TOOL_NO 1,BASE_NO 2,IPO_FRAME #BASE}
DECL PDAT PPDAT35={VEL 100.0,ACC 100.0,APO_DIST 100.0}
DECL E6POS XP35={x -84.1126785,y 889.032593,z 951.603394,a 53.6793785,b -33.1230698,c -50.1699104,s 6,t 19,e1 0.0,e2 0.0,e3 0.0,e4 0.0,e5 0.0,e6 0.0}
DECL FDAT FP35={TOOL_NO 1,BASE_NO 2,IPO_FRAME #BASE}
DECL PDAT PPDAT36={VEL 100.0,ACC 100.0,APO_DIST 100.0}
DECL E6POS XP36={x 336.611511,y 873.018677,z 811.395508,a 59.0088615,b -25.2084293,c -61.5601387,s 6,t 19,e1 0.0,e2 0.0,e3 0.0,e4 0.0,e5 0.0,e6 0.0}
DECL FDAT FP36={TOOL_NO 1,BASE_NO 2,IPO_FRAME #BASE}
DECL PDAT PPDAT37={VEL 100.0,ACC 100.0,APO_DIST 100.0}
DECL E6POS XP37={x 363.02771,y 1594.13403,z 616.088928,a 20.9962196,b 39.6207504,c -79.7914963,s 6,t 59,e1 0.0,e2 0.0,e3 0.0,e4 0.0,e5 0.0,e6 0.0}
DECL FDAT FP37={TOOL_NO 1,BASE_NO 2,IPO_FRAME #BASE}
DECL PDAT PPDAT38={VEL 100.0,ACC 100.0,APO_DIST 100.0}
DECL E6POS XP38={x 347.999298,y 2123.59204,z 1765.30701,a 7.69621086,b 41.4584999,c -132.413498,s 6,t 59,e1 0.0,e2 0.0,e3 0.0,e4 0.0,e5 0.0,e6 0.0}
DECL FDAT FP38={TOOL_NO 1,BASE_NO 2,IPO_FRAME #BASE}
DECL PDAT PPDAT39={VEL 100.0,ACC 100.0,APO_DIST 100.0}
DECL PDAT PPDAT40={VEL 100.0,ACC 100.0,APO_DIST 10.0}
ENDDAT
